// TIA Portal V17 export
// export: Created 2025-05-06T14:31:59.8182294Z, ExportSetting WithDefaults, DisplayName Totally Integrated Automation Portal, DisplayVersion V17 Update 8, DisplayName TIA Portal Openness, DisplayVersion V17 Update 8, DisplayName TIA Portal Version Control Interface, DisplayVersion V17, DisplayName SINAMICS Startdrive Advanced, DisplayVersion V17 SP2, DisplayName SINAMICS Startdrive G110M, G120, G120C, G120D, G120P, G115D, DisplayVersion V17 SP2, DisplayName SINAMICS Startdrive G130, G150, S120, S150, SINAMICS MV, S210, DisplayVersion V17 SP2, DisplayName STEP 7 Professional, DisplayVersion V17 Update 8, DisplayName SINUMERIK ONE STEP 7 Toolbox, DisplayVersion V17 Update 12, DisplayName SINUMERIK 840D sl STEP 7 Toolbox, DisplayVersion V17 Update 12, DisplayName STEP 7 Safety, DisplayVersion V17 Update 6, DisplayName WinCC Advanced, DisplayVersion V17 Update 8
DATA_BLOCK "DB10202_UNIT_2_PYROMETER"   // DB10202
{ DB_Accessible_From_OPC_UA := 'FALSE' }
AUTHOR : ETXETAR
VERSION : 1.0
// stored: AutoNumber false, DBAccessibleFromOPCUA false, DBAccessibleFromWebserver false, InstanceOfName FB10200_PYROMETERS, InstanceOfType FB
"FB10200_PYROMETERS"
   // VAR_INPUT
   //    OPTIONS_0 : Byte;
   //    DEVICE_STATUS_SENSOR_INPUT : Real;
   //    PROCESS_TEMP_SENSOR_INPUT : Real;
   //    HEAD_TEMP_SENSOR_INPUT : Real;
   //    T1_TEMP_SENSOR_INPUT : Real;
   //    T2_TEMP_SENSOR_INPUT : Real;
   //    CURRENT_EMISSIVITY_SENSOR_INPUT : Real;
   //    CURRENT_TRANSMISSION_SENSOR_INPUT : Real;
   //    UNIT_NUMBER : Int;
   // END_VAR
   // VAR_OUTPUT
   //    PROCESS_TEMP_LOW_WARNING : Bool;
   //    PROCESS_TEMP_HIGH_WARNING : Bool;
   //    PROCESS_TEMP_LOW_ALARM : Bool;
   //    PROCESS_TEMP_HIGH_ALARM : Bool;
   //    HEAD_TEMP_LOW_WARNING : Bool;
   //    HEAD_TEMP_HIGH_WARNING : Bool;
   //    HEAD_TEMP_LOW_ALARM : Bool;
   //    HEAD_TEMP_HIGH_ALARM : Bool;
   //    EMISSIVITY_LOW_WARNING : Bool;
   //    EMISSIVITY_HIGH_WARNING : Bool;
   //    EMISSIVITY_LOW_ALARM : Bool;
   //    EMISSIVITY_HIGH_ALARM : Bool;
   // END_VAR
   // VAR
   //    ANY_ACTIVE_ALARM : Bool;
   //    SEOC_ALARMS : Bool;
   //    RHP_SEOC_ALARMS : Bool;
   //    IS_SEOC_ALARMS : Bool;
   //    PROCESS_TEMP_SETTINGS : Struct
   //       LOW_WARNING_VALUE : Real;
   //       HIGH_WARNING_VALUE : Real;
   //       LOW_ALARM_VALUE : Real;
   //       HIGH_ALARM_VALUE : Real;
   //    END_STRUCT;
   //    HEAD_TEMP_SETTINGS : Struct
   //       LOW_WARNING_VALUE : Real;
   //       HIGH_WARNING_VALUE : Real;
   //       LOW_ALARM_VALUE : Real;
   //       HIGH_ALARM_VALUE : Real;
   //    END_STRUCT;
   //    EMISSIVITY_SETTINGS : Struct
   //       LOW_WARNING_VALUE : Real;
   //       HIGH_WARNING_VALUE : Real;
   //       LOW_ALARM_VALUE : Real;
   //       HIGH_ALARM_VALUE : Real;
   //    END_STRUCT;
   // END_VAR
BEGIN
END_DATA_BLOCK
